// TIA Portal V19 export
TYPE "LEXCHANGETRAY_typeNgStrapContronNodeMonitoring"
TITLE = exchangeTray_typeNgStrapContronNodeMonitoring
// exchangeTray_typeNgStrapContronNodeMonitoring related values
// stored: Access Published
   STRUCT
      simulated { ExternalAccessible := 'False'; ExternalVisible := 'False'; ExternalWritable := 'False'} : Bool;   // Simulation status
      signal { ExternalAccessible := 'False'; ExternalVisible := 'False'; ExternalWritable := 'False'} : Bool;   // Signal status
      error { ExternalAccessible := 'False'; ExternalVisible := 'False'; ExternalWritable := 'False'} : Bool;   // Error status
      countVal { ExternalAccessible := 'False'; ExternalVisible := 'False'; ExternalWritable := 'False'} : Int;   // Count value
   END_STRUCT;
END_TYPE
